FUNCTION_BLOCK NormallyOpenPushButton IMPLEMENTS I_PushButton
VAR
	input AT %I*	:	BOOL;
END_VAR

PROPERTY PUBLIC IsPressed : BOOL

// ho eliminato manualmente il Setter di questa proprietà perché qui non ha senso
GET
IsPressed := input;
END_GET
END_PROPERTY

PROPERTY PUBLIC IsReleased : BOOL

// ho eliminato manualmente il Setter di questa proprietà perché qui non ha senso
GET
IsReleased := NOT IsPressed;
END_GET
END_PROPERTY

END_FUNCTION_BLOCK

(* stored: Version 1.1.0.1, ProductVersion 3.1.4024.11
   POU NormallyOpenPushButton: Id {7bdd6fa5-3db6-4c9a-9599-965efae89c82}, SpecialFunc None
   Property IsPressed: Id {52879cf8-c77d-4907-ad83-011f48f68480}
   Get Get: Id {1d2a7500-d969-4f0b-ae30-dadbbc75aa92}
   Property IsReleased: Id {f84ce8d1-a934-45b7-ba38-b75ff545bcc4}
   Get Get: Id {f6404ceb-4163-4b07-85b9-e2c109cc6d59} *)
